% RSLogix 500 project TEST_OCT_21_2019_BAK000.RSS, saved by version 11.00.00.00 %
PROJECT "UNTITLED"    % processor: MicroLogix 1200 %

PROGRAM FILES
  LAD 2   8 rungs
  LAD 3, 4, 5, 6, 7, 8, 9, 10, 11, 12, 13, 14, 15: only END

DATA FILES
  O0 OUTPUT  4 elements
  I1 INPUT  4 elements
  S2 STATUS  66 elements
  B3 BINARY  32 elements
  T4 TIMER  40 elements
  C5 COUNTER  32 elements
  R6 CONTROL  16 elements
  N7 INTEGER  105 elements
  F8 FLOAT  1 elements

LADDER 2
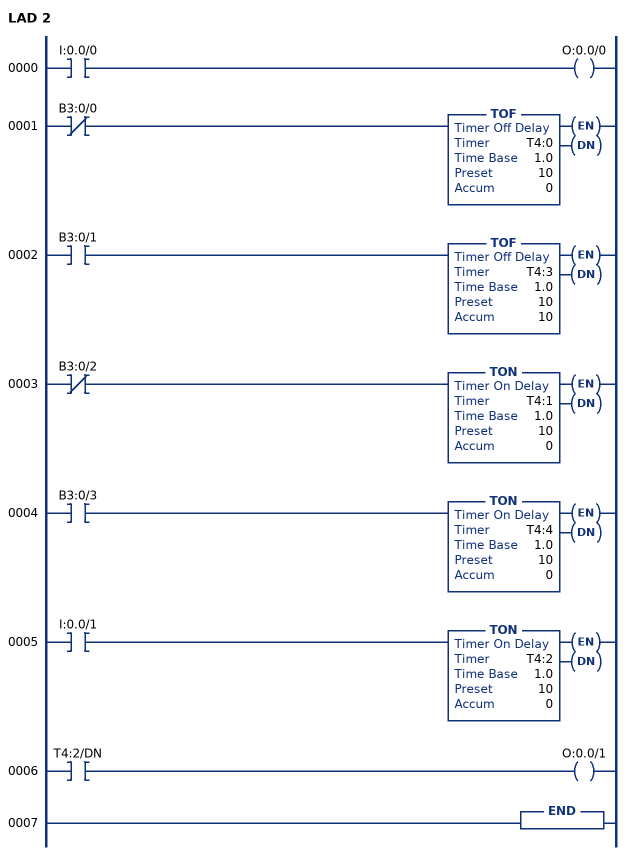
% Rung: 0 %
SOR XIC I:0.0/0 OTE O:0.0/0 EOR
% Rung: 1 %
SOR XIO B3:0/0 TOF T4:0 1.0 10 0 EOR
% Rung: 2 %
SOR XIC B3:0/1 TOF T4:3 1.0 10 10 EOR
% Rung: 3 %
SOR XIO B3:0/2 TON T4:1 1.0 10 0 EOR
% Rung: 4 %
SOR XIC B3:0/3 TON T4:4 1.0 10 0 EOR
% Rung: 5 %
SOR XIC I:0.0/1 TON T4:2 1.0 10 0 EOR
% Rung: 6 %
SOR XIC T4:2/DN OTE O:0.0/1 EOR
% Rung: 7 %
SOR END EOR

DATA TABLE (non-zero values as saved)
DATA B3
% B3:0 % 0X0004 0X0000 0X0000 0X0000 0X0000 0X0000 0X0000 0X0000 0X0000 0X0000
DATA T4
% .PRE .ACC %
% T4:0 % 10 0
% T4:1 % 10 0
% T4:2 % 10 0
% T4:3 % 10 10
% T4:4 % 10 0
